FUNCTION_BLOCK fb_exchangeTraySystem
VAR_IN_OUT
	var_ref_ele : ref_ele_io;
END_VAR
VAR_INPUT
	in_flg_run : BOOL;
	in_flg_start : BOOL;
	in_flg_pause : BOOL;
END_VAR
VAR_OUTPUT
	out_flg_run : BOOL;
	out_flg_busy : BOOL;
	out_flg_Done : BOOL;
	out_flg_error : BOOL;
END_VAR
VAR
	fbi_ele_controler: fb_ele_controller;
	var_buf_moveMode : eP_eleMoveMode;
	flg_run: BOOL;
END_VAR
VAR // added by the converter: edge detectors and wires of the graphical bodies
    _rt1 : R_TRIG;
    _ft1, _ft2 : F_TRIG;
    _w1 : BOOL;
END_VAR

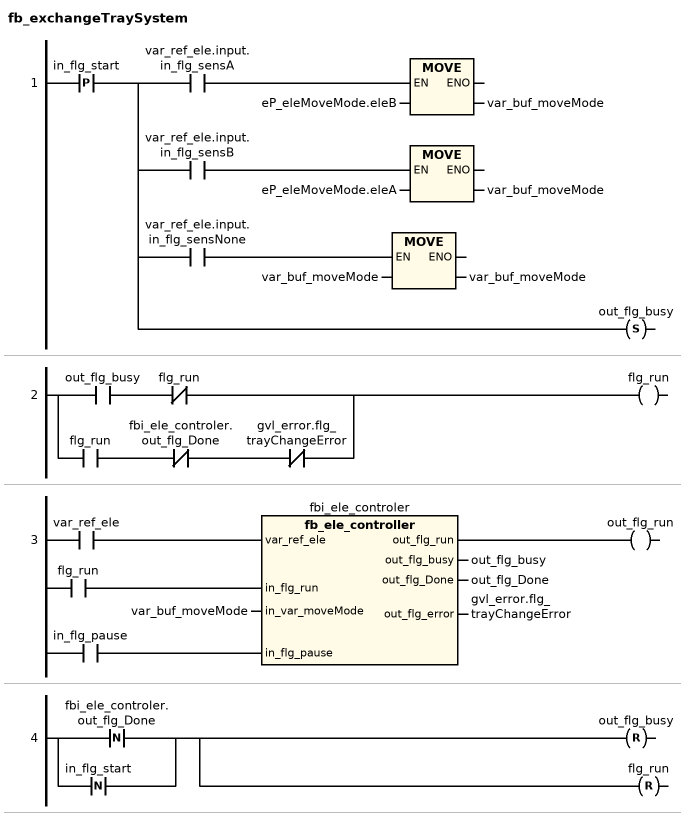
// NETWORK 1
_rt1(CLK := in_flg_start);
IF _rt1.Q AND var_ref_ele.input.in_flg_sensA THEN var_buf_moveMode := eP_eleMoveMode.eleB; END_IF
IF _rt1.Q AND var_ref_ele.input.in_flg_sensB THEN var_buf_moveMode := eP_eleMoveMode.eleA; END_IF
IF _rt1.Q AND var_ref_ele.input.in_flg_sensNone THEN var_buf_moveMode := var_buf_moveMode; END_IF
out_flg_busy S= _rt1.Q;

// NETWORK 2
flg_run := out_flg_busy AND NOT flg_run OR flg_run AND NOT fbi_ele_controler.out_flg_Done AND NOT gvl_error.flg_trayChangeError;

// NETWORK 3
fbi_ele_controler(
    var_ref_ele := var_ref_ele,
    in_flg_run := flg_run,
    in_var_moveMode := var_buf_moveMode,
    in_flg_pause := in_flg_pause,
    out_flg_busy => out_flg_busy,
    out_flg_Done => out_flg_Done,
    out_flg_error => gvl_error.flg_trayChangeError); // fb_ele_controller
out_flg_run := fbi_ele_controler.out_flg_run;

// NETWORK 4
_ft1(CLK := fbi_ele_controler.out_flg_Done);
_ft2(CLK := in_flg_start);
_w1 := _ft1.Q OR _ft2.Q;
out_flg_busy R= _w1;
flg_run R= _w1;

END_FUNCTION_BLOCK

(* stored: Version 1.1.0.1, ProductVersion 3.1.4024.11
   POU fb_exchangeTraySystem: Id {42579282-25e7-45b6-a140-1bb8eddccace}, SpecialFunc None *)
